DATA_BLOCK "DB_UnitTestControl"
{ S7_Optimized_Access := 'TRUE' }
VERSION : 0.1
NON_RETAIN
"STR_UnitTestControl"

BEGIN

END_DATA_BLOCK

